(* Schneider Machine Expert - Basic project POMPA RUN HOUR, file version 1.7.0.0 *)
(* ProjectInformations: Name=New project *)

HARDWARE
  Cpu 0: TM221M16R/G
  EthernetConfiguration: NetworkName=M221, IpAllocationMode=FixedAddress, IpAddress=0.0.0.0, SubnetMask=0.0.0.0
  SerialLineConfiguration: Baud=Baud19200, Parity=ParityEven, DataBits=DataBits8, StopBits=StopBits1, PhysicalMedium=PhysicalMediumRs485, TransmissionMode=TransmissionModeModbusRtu, SlaveId=1, Addressing=SlaveAddressing
  MastTask: UsePeriodScanMode=false, PeriodScan=100
  FastTask: Period=255
  CpuBehavior: StartingMode=StartAsPreviousState, AutoSaveRamOnEeprom=true, WatchdogPeriod=250

SYMBOLS  (address, symbol, comment, settings)
  %TM0        [Preset=5, Base=OneSecond]
  %TM1        [Preset=5, Base=OneSecond]
  %TM2        [Preset=10, Base=OneSecond, IsRetentive=true]
  %TM3        [Preset=10, Base=OneSecond, IsRetentive=true]
  %I0.1       "manual"
  %Q0.0       "P1"
  %Q0.1       "P2"

POU New POU
  (* SectionNumber=1 *)

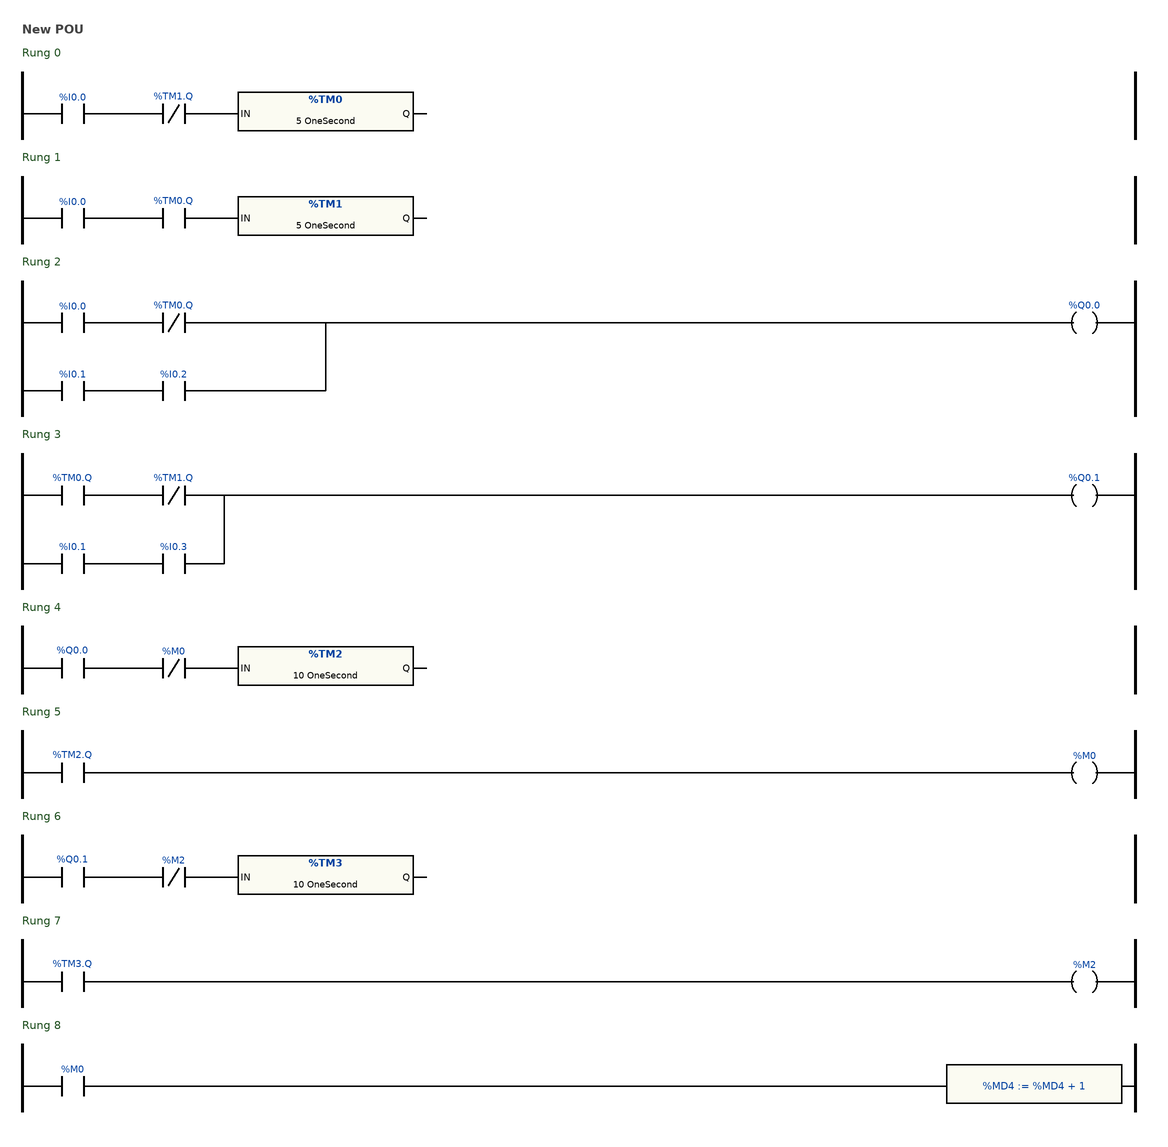

// Rung 0
  BLK %TM0
  LD %I0.0
  ANDN %TM1.Q
  IN
  END_BLK
  // as ST:
  //   %TM0(IN := %I0.0 AND NOT %TM1.Q);

// Rung 1
  BLK %TM1
  LD %I0.0
  AND %TM0.Q
  IN
  END_BLK
  // as ST:
  //   %TM1(IN := %I0.0 AND %TM0.Q);

// Rung 2
  LD %I0.0
  ANDN %TM0.Q
  OR( %I0.1
  AND %I0.2
  )
  ST %Q0.0
  // as ST:
  //   %Q0.0 := %I0.0 AND NOT %TM0.Q OR %I0.1 AND %I0.2;

// Rung 3
  LD %TM0.Q
  ANDN %TM1.Q
  OR( %I0.1
  AND %I0.3
  )
  ST %Q0.1
  // as ST:
  //   %Q0.1 := %TM0.Q AND NOT %TM1.Q OR %I0.1 AND %I0.3;

// Rung 4
  BLK %TM2
  LD %Q0.0
  ANDN %M0
  IN
  END_BLK
  // as ST:
  //   %TM2(IN := %Q0.0 AND NOT %M0);

// Rung 5
  LD %TM2.Q
  ST %M0
  // as ST:
  //   %M0 := %TM2.Q;

// Rung 6
  BLK %TM3
  LD %Q0.1
  ANDN %M2
  IN
  END_BLK
  // as ST:
  //   %TM3(IN := %Q0.1 AND NOT %M2);

// Rung 7
  LD %TM3.Q
  ST %M2
  // as ST:
  //   %M2 := %TM3.Q;

// Rung 8
  LD %M0
  [ %MD4 := %MD4 + 1 ]
  // as ST:
  //   IF %M0 THEN %MD4 := %MD4 + 1; END_IF;

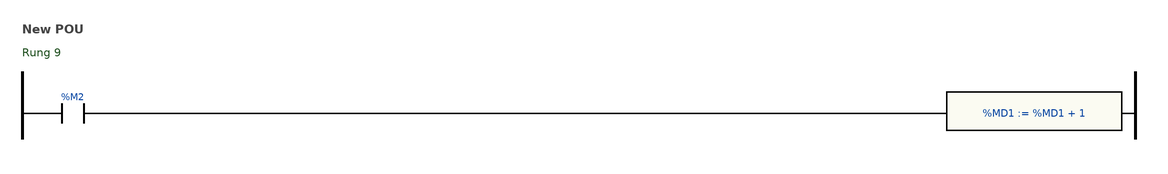

// Rung 9
  LD %M2
  [ %MD1 := %MD1 + 1 ]
  // as ST:
  //   IF %M2 THEN %MD1 := %MD1 + 1; END_IF;
